FUNCTION_BLOCK TRingCounter_INT
VAR
    Count : INT;
    _StartValue : INT;
    _EndValue : INT;
END_VAR

PROPERTY EndValue : INT
GET
EndValue := _EndValue;
END_GET
SET
_EndValue := EndValue;
END_SET
END_PROPERTY

METHOD FB_init : BOOL
VAR_INPUT
	bInitRetains : BOOL; // if TRUE, the retain variables are initialized (warm start / cold start)
	bInCopyCode : BOOL;  // if TRUE, the instance afterwards gets moved into the copy code (online change)

    StartValue : INT;
    EndValue : INT;
END_VAR
THIS^._StartValue := StartValue;
THIS^._EndValue := EndValue;
Reset();
END_METHOD

METHOD Inc
VAR_INPUT
END_VAR
Count := Count + 1;
IF Count > EndValue THEN
    Reset();
END_IF
END_METHOD

PROPERTY NextValue : INT
GET
IF Count = EndValue THEN
    NextValue := StartValue;
ELSE
    NextValue := Count + 1;
END_IF
END_GET
END_PROPERTY

METHOD Reset
VAR_INPUT
END_VAR
Count := StartValue;
END_METHOD

PROPERTY StartValue : INT
GET
StartValue := _StartValue;
END_GET
SET
_StartValue := StartValue;
END_SET
END_PROPERTY

PROPERTY Value : INT
GET
Value := Count;
END_GET
SET
Count := Value;
END_SET
END_PROPERTY

END_FUNCTION_BLOCK

(* stored: Version 1.1.0.1, ProductVersion 3.1.4024.3
   POU TRingCounter_INT: Id {8a8210f6-78b5-0e52-35a8-d458f4458b57}, SpecialFunc None
   Folder Methods: Id {b20cae32-0d3c-0a77-3a34-a15aefddb488}
   Folder Properties: Id {a95977ee-1d05-03eb-102a-8a7d47d5563d}
   Property EndValue: Id {9fa55c47-b7c8-0f79-330a-b802d766ecf0}
   Get Get: Id {86e2d56f-ea9a-093c-3711-bb886af6fb7f}
   Set Set: Id {d2342d71-9093-0f04-20d8-b39c3b97ec77}
   Method FB_init: Id {ae48539c-217e-082d-1915-d71ab05a4d01}
   Method Inc: Id {e4194c23-04f5-0360-2f2c-232d18402ffa}
   Property NextValue: Id {a99f870c-8d1e-069d-2f0d-fc9f0c7fe44b}
   Get Get: Id {6a09d59d-e204-0703-1be3-b2579699da08}
   Method Reset: Id {ecf49509-ee4c-0e01-3656-a7b72083a555}
   Property StartValue: Id {5cdbdd43-effb-0a63-0bd3-e32d3f9c3844}
   Get Get: Id {a77e0a3c-47cf-096d-3253-8730386a2966}
   Set Set: Id {61406e5a-35ed-0f50-1944-f3f04d44fdb3}
   Property Value: Id {3bc9b703-91fc-0298-3887-842936672537}
   Get Get: Id {2319fd5f-9959-0a8c-1162-1047ddfc53f2}
   Set Set: Id {0a82fea8-415b-0666-03eb-aa33c035daec} *)
